FUNCTION_BLOCK E_SWITCH
  (* Version 1.0, 2005-07-05, Goran Cengic, Chalmers *)
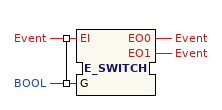
  EVENT_INPUT
    EI WITH G;
  END_EVENT
  EVENT_OUTPUT
    EO0;
    EO1;
  END_EVENT
  VAR_INPUT
    G : BOOL;
  END_VAR
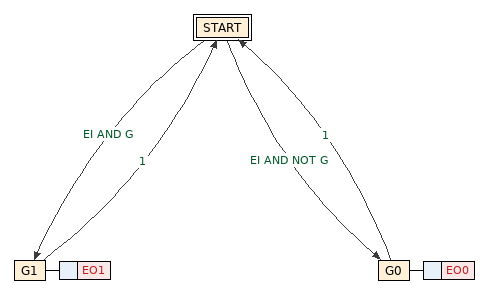
  EC_STATES
    START;
    G0 : -> EO0;
    G1 : -> EO1;
  END_STATES
  EC_TRANSITIONS
    START TO G0 := EI AND NOT G;
    G0 TO START := 1;
    START TO G1 := EI AND G;
    G1 TO START := 1;
  END_TRANSITIONS
END_FUNCTION_BLOCK
